// Mitsubishi GX Works2 project: PID   PLC: FX3G
// ПИД-регулятор Пример из видео

// global labels: Global1
VAR_GLOBAL
  AI_Pressure AT R100 : INT;
  xMode AT M500 : BOOL;
  xStart AT M501 : BOOL;
  xAT AT M502 : BOOL;
  xATMode AT M503 : BOOL;
  iSetValue AT R101 : INT;  (* Уставка - желаемое значение *)
  iDelta AT R103 : INT;
  xPump AT Y000 : BOOL;  (* Сигнал на запуск насоса *)
  iPumpTask AT R102 : INT;
END_VAR

// task Task_01 (event TRUE, interval 0, priority 31): POU_01
// user libraries (not included): AlarmManger128, Utils

PROGRAM POU_01
VAR
  fbHYST : HYST;
END_VAR
IF D8030 = 32760 THEN
		AI_Pressure :=0;
ELSE
		AI_Pressure := SCALE( D8030 , 0 , 4000 , 0 , 1000 );
END_IF;
	fbHYST(
	xIn:= (xStart AND NOT xMode) ,
	iSV:= iSetValue,
	iPV:= AI_Pressure ,
	iDV:= iDelta ,Q:= xPump
	 ); 
IF MEP(xStart) THEN 
		 R500 := 1000;
		 R501 := 2#0000_0000_0000_0001;
		 IF xAT AND xStart THEN 
			 	R501 := SETB( R501 , 4 );
			 	R501 := SETB( R501 , 5 );
			 	IF NOT xATMode THEN
			 			R51 := SETB( R501 , 6 );
			 	END_IF;
			 	xAT := FALSE;
		 END_IF;
		 R502 := 30;
		 R522 := 1000;
		 R523 := 0;
		 R525 := iDelta;
		 R526 := R522;
		 R527 := R523;
END_IF;
PID( 
(xStart AND NOT xMode) , 
iSetValue, 
AI_Pressure, 
R500, 
iPumpTask 
);
END_PROGRAM
